FUNCTION_BLOCK SAMPLE_4 (* 4-variable sampling-See SAMPLE_1 for sequences *)
  (* Standard: 61499-1; Function: Sampling; Type: 4-variable *)
  (* Version 0.0, 2002-02-15, JHC, Rockwell Automation *)
  (* Compiler header: package fb.rt.math; *)
  (* Compiler Java IBM VisualAge 3.0 *)
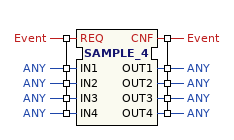
  EVENT_INPUT
    REQ WITH IN1, IN2, IN3, IN4; (* Request to Sample with Monitor Lock *)
  END_EVENT
  EVENT_OUTPUT
    CNF WITH OUT1, OUT2, OUT3, OUT4; (* Initial Sample or OUT1 changed *)
  END_EVENT
  VAR_INPUT
    IN1 : ANY; (* Data to Sample *)
    IN2 : ANY;
    IN3 : ANY;
    IN4 : ANY;
  END_VAR
  VAR_OUTPUT
    OUT1 : ANY; (* Sampled Data *)
    OUT2 : ANY;
    OUT3 : ANY;
    OUT4 : ANY;
  END_VAR
END_FUNCTION_BLOCK
